{attribute 'linkalways'}
{attribute 'hide_all_locals'}
FUNCTION_BLOCK ValueUlintRead EXTENDS ValueBase IMPLEMENTS ValueRead
VAR
	thisValue : ULINT;
END_VAR

{attribute 'call_after_global_init_slot' := '1'}
{attribute 'call_after_online_change_slot' := '1'}
METHOD PROTECTED GetThisAnyType
VAR_INPUT
END_VAR
thisAnyType := ToAnyType(thisValue);
END_METHOD

METHOD GetAsType : BOOL
VAR_INPUT
	destination : __SYSTEM.AnyType;
END_VAR
GetAsType := ConvertAnyType(thisAnyType, destination);
END_METHOD

METHOD GetAsString : T_MaxString
VAR_INPUT
END_VAR
GetAsString := TO_STRING(thisValue);
END_METHOD

METHOD Get : BOOL
VAR_INPUT
	destination : ANY;
END_VAR
Get := ConvertAnyType(thisAnyType, destination);
END_METHOD

METHOD FB_init : BOOL
VAR_INPUT
	bInitRetains : BOOL; // if TRUE, the retain variables are initialized (warm start / cold start)
	bInCopyCode : BOOL;  // if TRUE, the instance afterwards gets moved into the copy code (online change)
END_VAR
_ValueType := __SYSTEM.TYPE_CLASS.TYPE_ULINT;
END_METHOD

{attribute 'monitoring' := 'call'}
PROPERTY Value : ULINT
GET
Value := thisValue;
END_GET
END_PROPERTY

END_FUNCTION_BLOCK

(* stored: Version 1.1.0.1
   POU ValueUlintRead: Id {911ac8c1-62d5-48d6-a4c5-b248d5eb5053}, SpecialFunc None
   Method GetThisAnyType: Id {e1864f38-81f9-44f5-99be-5aac3b9337d9}
   Method GetAsType: Id {c12deb2b-f173-4cec-992e-512d4f2f87db}
   Method GetAsString: Id {c0b4c72f-6707-439d-9628-b3cff05cb3a4}
   Method Get: Id {247be177-5b4e-49f7-805f-7546d6ff5e6b}
   Method FB_init: Id {7017282d-832b-4f7b-8577-f23003959141}
   Property Value: Id {37b93a4e-bf04-493a-ac01-1194f093691a}
   Get Get: Id {cdcb8aa8-9963-4eb7-b5bd-36c79ac576d5} *)
